// TIA Portal V19 export
FUNCTION "AnalogWritingSystem" : Void   // FC13, STL
TITLE = ANALOG OUTPUT: CONVERT FROM mA TO PAW VALUE
{ S7_Optimized_Access := 'TRUE' }
AUTHOR : FLA
FAMILY : UHT
VERSION : 1.0
// Programmer Init: 8953-FLA
// 
// Change Log:
// 
// Date        Change                          Updated by
// ------------------------------------------------------
// 19.04.99    1. Edition                      FLA
// stored: AutoNumber false
   VAR_INPUT
      OUT_VAL : Int;
      MIN_REAL : Real;
      MAX_REAL : Real;
   END_VAR
   VAR_OUTPUT
      OUT_DA_CONV : Word;
   END_VAR
   VAR_TEMP
      SPAN : Real;
   END_VAR
BEGIN

NETWORK
TITLE = CONVERT FROM mA TO PAW VALUE
// Comment
      L     #MAX_REAL;  // max output
      L     #MIN_REAL;  // min output
      -R;
      T     #SPAN;  // output span
      L     #OUT_VAL;  // mA from regulator
      ITD;
      DTR;
      L     #MIN_REAL;
      -R;
      L     1000.0;
      *R;
      L     #SPAN;
      /R;
      L     27648.0;
      *R;
      L     1000.0;
      /R;
      RND+;
      T     #OUT_DA_CONV;  // output to analog card
END_FUNCTION
